Yaskawa INFORM job: SKRZYNIA_5040_180_STOPNI_10BR.JBI

/JOB
//NAME SKRZYNIA_5040_180_STOPNI_10BR
///FOLDERNAME 02-SKRZYNIE_JOBS
//POS
///NPOS 329,329,0,22,0,0
///TOOL 0
///POSTYPE PULSE
///PULSE
C00000=-21231,-51303,42314,2367,6591,-1439
C00001=-12854,-61498,-6635,149088,-29435,16513
C00002=84284,-61498,-6635,149088,14842,16513
C00003=84426,-61498,-62039,149088,14842,16513
C00004=84426,-61498,-83719,149088,14842,16513
C00005=79414,-27317,-83719,149088,18958,2543
C00006=69654,-19285,-77591,161600,-10201,-10832
C00007=70169,-17945,-76482,160305,-10504,-10321
C00008=68101,-15975,-74811,167053,-10620,-13110
C00009=69917,-14828,-73813,161695,-10968,-10930
C00010=70169,-17945,-76482,160305,-10504,-10321
C00011=40079,-25830,-61904,72398,37828,17494
C00012=40079,-25830,-61904,72398,37828,17494
C00013=38824,-23395,-60038,72349,38727,17731
C00014=41545,-22667,-59464,70826,37145,18191
C00015=40079,-25830,-61904,72398,37828,17494
C00016=62247,-7095,-69897,102362,7855,12255
C00017=53704,-22919,-41820,136356,29967,-7241
C00018=40577,-31455,-39147,101508,36831,1521
C00019=40669,-23760,-31845,100563,36582,2074
C00020=41101,-23552,-31684,100574,36285,2055
C00021=39898,-21530,-30092,99854,36985,2518
C00022=41920,-21198,-29826,100065,35629,2328
C00023=41101,-23552,-31684,100574,36285,2055
C00024=40577,-31455,-39147,101508,36831,1521
C00025=45746,-39048,-62846,85420,33792,9363
C00026=93007,-60609,-51405,156585,32340,-40977
C00027=83918,-61953,-48743,149551,29621,-25735
C00028=40577,-31455,-39147,101508,36831,1521
C00029=63645,-11488,-68603,127053,9270,213
C00030=57886,960,-43515,148211,29579,-11223
C00031=58100,6617,-53508,135301,20179,-4597
C00032=58076,11581,-47409,136064,20541,-4974
C00033=56683,13582,-44848,135736,21192,-4491
C00034=57911,14088,-44192,136506,20851,-5156
C00035=58076,11581,-47409,136064,20541,-4974
C00036=58100,6617,-53508,135301,20179,-4597
C00037=57886,960,-43515,148211,29579,-11223
C00038=63645,-11488,-68603,127053,9270,213
C00039=46424,-32589,-51504,107545,30005,2440
C00040=46670,-25209,-46239,104499,29210,4073
C00041=45428,-23318,-44777,103595,29873,4669
C00042=46971,-23118,-44620,103792,28881,4430
C00043=46670,-25209,-46239,104499,29210,4073
C00044=44789,-32224,-51260,106964,30993,2875
C00045=42092,-32720,-44065,59648,38266,12707
C00046=43496,-26383,-41044,56137,38810,14761
C00047=42389,-24633,-39725,56307,39660,14725
C00048=44413,-24250,-39432,55137,38557,15308
C00049=43496,-26383,-41044,56137,38810,14761
C00050=44564,-32742,-56962,40463,46428,19920
C00051=40345,-33419,-45947,59645,39680,12787
C00052=90538,-65158,-52413,145953,6697,-22013
C00053=90538,-65158,-52413,145953,6697,-22013
C00054=86028,-64310,-60026,34123,6588,25352
C00055=40577,-31455,-39147,101508,36831,1521
C00056=59968,-20268,-35682,154489,33643,-14406
C00057=58485,-14292,-30532,152791,33122,-13346
C00058=56876,-12305,-28713,151388,33319,-12442
C00059=58661,-11495,-27956,152741,32764,-13330
C00060=58485,-14292,-30532,152791,33122,-13346
C00061=59968,-20268,-35682,154489,33643,-14406
C00062=40577,-31455,-39147,101508,36831,1521
C00063=40577,-27956,-24714,110033,39226,-3600
C00064=40832,-22290,-20525,108598,38533,-2722
C00065=39477,-20111,-18797,107655,39231,-2172
C00066=41591,-19772,-18521,108272,37862,-2511
C00067=40832,-22290,-20525,108598,38533,-2722
C00068=40577,-31455,-39147,101508,36831,1521
C00069=86028,-64310,-60026,34123,6588,25352
C00070=86028,-64310,-60026,57978,24772,25352
C00071=86028,-64309,-60028,57978,24769,25352
C00072=40577,-31455,-39147,101508,36831,1521
C00073=40577,-31455,-39147,101508,36831,1521
C00074=41094,-24086,-28510,103808,36979,148
C00075=39566,-21578,-26552,102813,37826,761
C00076=41385,-20827,-24026,104651,36978,-353
C00077=41094,-24086,-28510,103808,36979,148
C00078=37787,-19718,1186,119438,46446,-9893
C00079=45975,-24882,-879,104701,32906,-9183
C00080=73009,-53529,-38439,45960,15190,15723
C00081=45844,-59376,-6382,28358,16063,-8083
C00082=0,-52280,40443,0,6876,0
C00083=-681,-52632,38645,-5695,5489,-631
C00084=-17840,-61498,-6635,-149088,-29435,-16513
C00085=-84284,-61498,-6635,-149088,14842,-16513
C00086=-84426,-61498,-62039,-149088,14842,-16513
C00087=-84426,-61498,-83719,-149088,14842,-16513
C00088=-79414,-27317,-83719,-149088,18958,-2543
C00089=-69654,-19285,-77591,-161600,-10201,10832
C00090=-70169,-17945,-76482,-160305,-10504,10321
C00091=-68828,-16679,-75416,-164694,-10564,12135
C00092=-70730,-15407,-74323,-159180,-10987,9897
C00093=-70169,-17945,-76482,-160305,-10504,10321
C00094=-69654,-19285,-77591,-161600,-10201,10832
C00095=-79414,-27317,-83719,-149088,18958,-2543
C00096=-79414,-27317,-83719,-149088,18958,-2543
C00097=-83351,-27062,-60322,-167360,37385,6517
C00098=-83351,-27062,-60322,-167360,37385,23281
C00099=-45097,-23850,-79932,-76262,26943,-22849
C00100=-48253,-15729,-73342,-71138,25693,-24842
C00101=-50302,-13076,-73239,-65836,25323,-27140
C00102=-49401,-11675,-71961,-66260,25816,-27133
C00103=-50608,-11574,-71867,-65226,25249,-27391
C00104=-49660,-13361,-73494,-66442,25615,-26975
C00105=-48242,-21102,-77802,-73044,25430,-23851
C00106=-42432,-29691,-46140,-101591,34194,-3953
C00107=-39561,-32409,-42051,-71473,38885,-9254
C00108=-41445,-24166,-34417,-69795,37942,-10196
C00109=-41357,-25431,-35380,-70168,37910,-9978
C00110=-40141,-23420,-33843,-70026,38836,-10113
C00111=-41944,-23213,-33680,-69384,37685,-10425
C00112=-41357,-25431,-35380,-70168,37910,-9978
C00113=-39561,-32409,-42051,-71473,38885,-9254
C00114=-81019,-65479,-53594,-111483,16801,11860
C00115=-83918,-61953,-48743,-149551,29621,25735
C00116=-40577,-31455,-39147,-101508,36831,-1521
C00117=-49519,-25509,-75942,-81549,24001,-19130
C00118=-42138,-12822,-51897,-114220,37124,-2825
C00119=-42418,-8239,-63642,-99180,32968,-11424
C00120=-44218,-2315,-57613,-98259,31965,-11515
C00121=-43448,-826,-56017,-98426,32361,-11601
C00122=-45030,-456,-55613,-98008,31536,-11462
C00123=-44218,-2315,-57613,-98259,31965,-11515
C00124=-42418,-8239,-63642,-99180,32968,-11424
C00125=-46424,-32589,-51504,-107545,30005,-2440
C00126=-47664,-24599,-45775,-104463,28531,-3999
C00127=-46974,-23582,-44988,-103952,28901,-4330
C00128=-48737,-23213,-44698,-104162,27760,-4069
C00129=-47664,-24599,-45775,-104463,28531,-3999
C00130=-44789,-32224,-51260,-106964,30993,-2875
C00131=-52916,-26599,-39279,-28650,42861,-21372
C00132=-54590,-19092,-33239,-26753,43640,-22510
C00133=-53867,-18183,-32472,-27186,44006,-22274
C00134=-55270,-17868,-32204,-26176,43615,-22844
C00135=-54590,-19092,-33239,-26753,43640,-22510
C00136=-51388,-27442,-41316,-29309,44045,-21030
C00137=-62081,-38823,-47091,-30795,32483,-22364
C00138=-86028,-64310,-60024,-34123,6590,-25350
C00139=-86028,-64310,-60026,-34123,6588,-25352
C00140=-86028,-64310,-60026,-34123,6588,-25352
C00141=-40577,-31455,-39147,-101508,36831,-1521
C00142=-46190,-29637,-41119,-118468,33777,2449
C00143=-49093,-22876,-34875,-118816,31686,2771
C00144=-47416,-20516,-32984,-117411,32403,1908
C00145=-48747,-20402,-32891,-117991,31622,2296
C00146=-49093,-22876,-34875,-118816,31686,2771
C00147=-46494,-29071,-39687,-120554,34221,3238
C00148=-39561,-32409,-42051,-71473,38885,-9254
C00149=-39561,-29125,-27808,-80306,37382,-3940
C00150=-43436,-23752,-23915,-78119,34960,-5282
C00151=-41521,-20874,-21664,-77573,36353,-5586
C00152=-43032,-20790,-21597,-77323,35339,-5740
C00153=-43436,-23752,-23915,-78119,34960,-5282
C00154=-39561,-32409,-42051,-71473,38885,-9254
C00155=-86028,-64310,-60026,-34123,6588,-25352
C00156=-86028,-64310,-60026,-57978,24772,-25352
C00157=-86028,-64309,-60028,-57978,24769,-25352
C00158=-40577,-28664,-27343,-108630,38732,2744
C00159=-40577,-31455,-39147,-101508,36831,-1521
C00160=-43516,-21710,-22385,-107479,36200,2021
C00161=-42168,-19388,-19611,-107236,37117,1884
C00162=-43632,-19706,-21236,-106626,35874,1517
C00163=-43516,-21710,-22385,-107479,36200,2021
C00164=-37787,-19718,1186,-119438,46446,9893
C00165=-42073,-20304,2487,-100625,34839,7554
C00166=-73009,-40277,-6382,-95546,11240,8083
C00167=-45844,-59376,-6382,-28358,16063,8083
C00168=0,-52280,40443,0,6876,0
C00169=0,-52280,40443,0,6876,0
C00170=0,-52280,40443,0,6876,0
C00171=17840,-61498,-6635,149088,-29435,16513
C00172=84284,-61498,-6635,149088,14842,16513
C00173=84426,-61498,-62039,149088,14842,16513
C00174=84426,-61498,-83719,149088,14842,16513
C00175=79414,-27317,-83719,149088,18958,2543
C00176=69654,-19285,-77591,161600,-10201,-10832
C00177=76421,-10554,-96109,158804,-42582,-3780
C00178=72151,-15398,-68153,108866,-8938,34672
C00179=72146,-15003,-68876,113258,-9266,32587
C00180=76421,-10554,-96109,158804,-42582,-3780
C00181=34693,-20653,-55351,82826,43754,17424
C00182=36026,-17403,-55626,79704,43213,19225
C00183=36110,-16271,-60816,75273,43939,22119
C00184=33117,-22954,-57201,83762,44711,17076
C00185=44072,-25282,-29267,59074,37137,11149
C00186=35613,-12237,-16796,64347,49532,7989
C00187=35669,-10629,-9632,67221,48090,5904
C00188=43298,-18069,-12230,66933,34938,6545
C00189=45101,-28611,-34216,51905,38288,13313
C00190=86972,-59792,-47806,52261,11911,13502
C00191=84284,-61498,-6635,149088,14842,16513
C00192=17840,-61498,-6635,149088,-29435,16513
C00193=0,-52280,40443,0,6876,0
C00194=-84284,-61498,-6635,-149088,14842,-16513
C00195=-84426,-61498,-62039,-149088,14842,-16513
C00196=-34728,-20635,-55362,-82794,43735,-17439
C00197=-36397,-18395,-56469,-79733,42961,-19136
C00198=-36362,-17151,-61599,-75273,43766,-22060
C00199=-33152,-22936,-57213,-83730,44691,-17092
C00200=-40586,-30782,-66310,-80775,34854,-15242
C00201=-40692,-30585,-47134,-93878,35604,-6100
C00202=-40870,-31947,-42232,-63836,39356,-11267
C00203=-40932,-24208,-34937,-62959,39653,-11802
C00204=-45435,-25401,-38781,-45915,41942,-16635
C00205=-39287,-15996,-33256,-50997,52191,-14482
C00206=-39287,-15215,-27013,-53302,49993,-12721
C00207=-47238,-24614,-37591,-45025,40897,-17096
C00208=-47977,-29416,-47116,-37884,44778,-19458
C00209=-89911,-63274,-62690,-19483,20389,-28477
C00210=-84284,-61498,-6635,-149088,14842,-16513
C00211=-17840,-61498,-6635,-149088,-29435,-16513
C00212=-2124,-53377,34839,-17747,2554,-1966
C00213=0,-52279,40442,0,6873,-1
C00214=65212,-60046,-8049,104848,-4690,-17864
C00215=40577,-31455,-39147,101508,36831,1521
C00216=38935,-8667,-59866,96806,37491,11641
C00217=39872,-3948,-62200,89905,36425,15493
C00218=40123,-1398,-59509,89712,36292,15545
C00219=40076,1432,-63122,83669,36365,19101
C00220=39872,-3948,-62200,89905,36425,15493
C00221=38788,-10415,-65666,93500,37192,13644
C00222=38494,-13737,-58620,102504,38775,8306
C00223=46486,-25212,-81916,68038,29584,25152
C00224=40809,-36068,-61713,64442,39202,15742
C00225=42276,-26166,-36634,93086,33999,4511
C00226=42397,-24236,-35180,92449,33874,4870
C00227=42456,-24928,-41878,86540,33672,8224
C00228=42276,-26166,-36634,93086,33999,4511
C00229=39142,-35579,-61405,65081,40271,15536
C00230=56371,-25371,-52824,18615,54374,25524
C00231=56370,-25165,-46553,19645,50450,24711
C00232=56832,-16031,-39063,18899,51967,25222
C00233=56804,-15583,-32487,20072,48035,24353
C00234=56370,-25165,-46553,19645,50450,24711
C00235=57699,-31993,-47488,30685,42383,20627
C00236=72028,-54906,-32140,129304,10545,-19932
C00237=68553,-57528,-19846,116818,2770,-18873
C00238=80051,-74607,19733,-8233,-9721,30787
C00239=0,-52279,40442,0,6873,1
C00240=-65212,-60046,-8049,-104848,-4690,17864
C00241=-65212,-60046,-8049,-104848,-4690,17864
C00242=-38865,-30967,-34224,-83703,38027,-4479
C00243=-46136,-6939,-46632,-121706,34309,84
C00244=-46867,-3267,-49648,-115679,31344,-3160
C00245=-48114,-333,-46510,-115722,30691,-2892
C00246=-48219,1611,-50657,-109137,28744,-6443
C00247=-46867,-3267,-49648,-115679,31344,-3160
C00248=-46241,-9247,-52869,-118634,32829,-1638
C00249=-45976,-11042,-44788,-126297,37070,2732
C00250=-52833,-24736,-69580,-100186,20368,-10781
C00251=-41290,-34357,-47396,-89099,34671,-6127
C00252=-41655,-21075,-14083,-101384,36064,2719
C00253=-43548,-19389,-12736,-101518,34735,2718
C00254=-43554,-21360,-20853,-95828,33898,-537
C00255=-41655,-21075,-14083,-101384,36064,2719
C00256=-39902,-32831,-41704,-71274,37363,-9142
C00257=-59997,-20337,-29256,-15458,45038,-24823
C00258=-49653,-28135,-37805,-37523,39695,-18391
C00259=-43199,-13906,-27547,-44351,51052,-15347
C00260=-43351,-12703,-20152,-46774,48118,-13551
C00261=-49653,-28135,-37805,-37523,39695,-18391
C00262=-55865,-33769,-26948,-46240,25044,-14477
C00263=-87889,-52133,-21276,-78165,-5410,-1028
C00264=0,-52279,40442,0,6873,1
C00265=1,-52278,40440,0,6869,2
C00266=71244,-62242,-42760,28259,6636,20995
C00267=86028,-64310,-60026,34123,6588,25352
C00268=40577,-31455,-39147,101508,36831,1521
C00269=59968,-20268,-35682,154489,33643,-14406
C00270=58485,-13865,-27025,153905,35067,-13980
C00271=58455,-11202,-24562,153724,34784,-13877
C00272=58575,-12016,-31397,151462,30972,-12614
C00273=58485,-13865,-27025,153905,35067,-13980
C00274=59968,-20268,-35682,154489,33643,-14406
C00275=40577,-31455,-39147,101508,36831,1521
C00276=39533,-29159,-27906,80257,37406,3969
C00277=37605,-21741,-8857,99005,39903,-3768
C00278=39778,-16633,-4738,98441,38266,-3268
C00279=39778,-19203,-13530,93410,37627,-246
C00280=39876,-23449,-23758,78420,37382,5067
C00281=40577,-31455,-39147,101508,36831,1521
C00282=86028,-64310,-60026,34123,6588,25352
C00283=71244,-62242,-42760,28259,6636,20995
C00284=1,-52278,40440,0,6869,2
C00285=1,-52278,40440,0,6869,2
C00286=-71244,-62242,-42760,-28259,6636,-20995
C00287=-86028,-64310,-60026,-34123,6588,-25352
C00288=-40577,-31455,-39147,-101508,36831,-1521
C00289=-59968,-20268,-35682,-154489,33643,14406
C00290=-58485,-13865,-27025,-153905,35067,13980
C00291=-60457,-10469,-23870,-155260,34234,14880
C00292=-60514,-11164,-30597,-153048,30384,13645
C00293=-58485,-13865,-27025,-153905,35067,13980
C00294=-59968,-20268,-35682,-154489,33643,14406
C00295=-40577,-31455,-39147,-101508,36831,-1521
C00296=-39561,-29149,-27902,-80249,37387,-3974
C00297=-37632,-21733,-8858,-99006,39884,3767
C00298=-42115,-16101,-4294,-98986,36705,3442
C00299=-42200,-18704,-13124,-93672,35977,314
C00300=-39902,-23438,-23752,-78411,37365,-5072
C00301=-39561,-32409,-42051,-71473,38885,-9254
C00302=-86028,-64310,-60026,-34123,6588,-25352
C00303=-71244,-62242,-42760,-28259,6636,-20995
C00304=-1,-52278,40440,0,6869,-2
C00305=2,-52272,40438,1,6859,6
C00306=86028,-64309,-60028,57978,24769,25352
C00307=40577,-31455,-39147,101508,36831,1521
C00308=41094,-22734,-22712,107351,37942,-1964
C00309=41295,-19722,-19354,107466,37828,-2032
C00310=41253,-21899,-28956,101408,36344,1561
C00311=41094,-22306,-21006,108327,38251,-2553
C00312=37787,-19718,1186,119438,46446,-9893
C00313=73009,-40734,-7449,93649,11189,-7175
C00314=45844,-59376,-6382,28358,16063,-8083
C00315=0,-52280,40443,0,6876,0
C00316=-2,-52272,40438,-1,6859,-6
C00317=-86028,-64309,-60028,-57978,24769,-25352
C00318=-40577,-30748,-35855,-103638,37302,-257
C00319=-40400,-24560,-25747,-102945,37769,566
C00320=-40181,-24927,-30789,-96759,37058,-2330
C00321=-42523,-20980,-24961,-98936,35699,-1187
C00322=-42523,-22298,-31586,-94154,35106,-3962
C00323=-42312,-27031,-36420,-94462,35277,-3790
C00324=-37787,-19718,1186,-119438,46446,9893
C00325=-73009,-37989,-1068,-104580,11683,12408
C00326=-45844,-59376,-6382,-28358,16063,8083
C00327=0,-52280,40443,0,6876,0
C00328=0,-52279,40442,1,6873,0
BC00000=467225
BC00001=513669
BC00002=494109
BC00003=467540
BC00004=467540
BC00005=467540
BC00006=467540
BC00007=467540
BC00008=467540
BC00009=467540
BC00010=467540
BC00011=478876
BC00012=478876
BC00013=478876
BC00014=478876
BC00015=478876
BC00016=566479
BC00017=516375
BC00018=516375
BC00019=516375
BC00020=516375
BC00021=516375
BC00022=516375
BC00023=516375
BC00024=516375
BC00025=488496
BC00026=488496
BC00027=675626
BC00028=675626
BC00029=717870
BC00030=717870
BC00031=717870
BC00032=717870
BC00033=717870
BC00034=717870
BC00035=717870
BC00036=717870
BC00037=717870
BC00038=717870
BC00039=686402
BC00040=686402
BC00041=686402
BC00042=686402
BC00043=686402
BC00044=686402
BC00045=673769
BC00046=686402
BC00047=686402
BC00048=686402
BC00049=686402
BC00050=686402
BC00051=641577
BC00052=641414
BC00053=760541
BC00054=849627
BC00055=849627
BC00056=849627
BC00057=849627
BC00058=849627
BC00059=849627
BC00060=849627
BC00061=849627
BC00062=849627
BC00063=849627
BC00064=849627
BC00065=849627
BC00066=849627
BC00067=849627
BC00068=849627
BC00069=849627
BC00070=849627
BC00071=998332
BC00072=998017
BC00073=1002378
BC00074=995834
BC00075=995834
BC00076=993496
BC00077=995834
BC00078=965704
BC00079=965704
BC00080=965704
BC00081=879640
BC00082=828403
BC00083=518986
BC00084=509920
BC00085=467540
BC00086=467540
BC00087=467540
BC00088=467540
BC00089=467540
BC00090=467540
BC00091=467540
BC00092=467540
BC00093=467540
BC00094=467540
BC00095=467540
BC00096=550011
BC00097=521167
BC00098=520352
BC00099=535759
BC00100=535759
BC00101=535757
BC00102=535757
BC00103=535757
BC00104=535757
BC00105=535757
BC00106=485653
BC00107=485653
BC00108=485653
BC00109=485653
BC00110=485653
BC00111=485653
BC00112=485653
BC00113=485653
BC00114=485653
BC00115=675626
BC00116=675626
BC00117=687148
BC00118=687148
BC00119=687148
BC00120=687148
BC00121=687148
BC00122=687148
BC00123=687148
BC00124=687148
BC00125=686402
BC00126=686401
BC00127=686401
BC00128=686401
BC00129=686401
BC00130=686402
BC00131=655680
BC00132=655680
BC00133=655680
BC00134=655680
BC00135=655680
BC00136=655680
BC00137=643721
BC00138=659181
BC00139=817027
BC00140=849627
BC00141=849627
BC00142=818905
BC00143=818905
BC00144=818905
BC00145=818905
BC00146=818905
BC00147=818905
BC00148=818905
BC00149=818905
BC00150=818905
BC00151=818905
BC00152=818905
BC00153=818905
BC00154=818905
BC00155=849627
BC00156=849627
BC00157=983499
BC00158=985574
BC00159=996021
BC00160=990664
BC00161=989585
BC00162=991221
BC00163=990664
BC00164=965704
BC00165=965704
BC00166=946312
BC00167=879640
BC00168=828403
BC00169=639407
BC00170=514217
BC00171=512528
BC00172=467540
BC00173=467540
BC00174=467540
BC00175=467540
BC00176=467540
BC00177=467540
BC00178=467538
BC00179=467538
BC00180=467540
BC00181=489674
BC00182=489674
BC00183=489674
BC00184=489674
BC00185=454931
BC00186=454931
BC00187=454931
BC00188=454931
BC00189=454931
BC00190=454931
BC00191=467540
BC00192=515629
BC00193=504733
BC00194=467540
BC00195=467540
BC00196=489675
BC00197=489675
BC00198=489675
BC00199=489675
BC00200=489675
BC00201=477973
BC00202=477973
BC00203=477973
BC00204=462612
BC00205=462612
BC00206=462612
BC00207=462612
BC00208=462612
BC00209=462612
BC00210=467540
BC00211=497858
BC00212=502748
BC00213=574255
BC00214=557840
BC00215=654869
BC00216=687148
BC00217=687148
BC00218=687148
BC00219=687148
BC00220=687148
BC00221=687148
BC00222=687148
BC00223=687148
BC00224=655680
BC00225=655680
BC00226=655680
BC00227=655680
BC00228=655680
BC00229=655680
BC00230=655680
BC00231=655680
BC00232=655680
BC00233=655680
BC00234=655680
BC00235=638520
BC00236=608041
BC00237=573428
BC00238=574255
BC00239=574255
BC00240=626137
BC00241=536464
BC00242=650227
BC00243=687148
BC00244=687148
BC00245=687148
BC00246=687148
BC00247=687148
BC00248=687148
BC00249=687148
BC00250=687148
BC00251=655680
BC00252=624958
BC00253=624958
BC00254=624958
BC00255=624958
BC00256=624958
BC00257=624958
BC00258=655680
BC00259=655680
BC00260=655680
BC00261=655680
BC00262=605110
BC00263=576379
BC00264=574255
BC00265=574254
BC00266=802302
BC00267=849627
BC00268=849627
BC00269=849627
BC00270=849627
BC00271=849627
BC00272=849627
BC00273=849627
BC00274=849627
BC00275=849627
BC00276=818905
BC00277=818905
BC00278=818905
BC00279=818905
BC00280=818905
BC00281=849627
BC00282=849627
BC00283=802302
BC00284=652677
BC00285=652677
BC00286=802302
BC00287=849627
BC00288=849627
BC00289=849627
BC00290=849627
BC00291=849629
BC00292=849627
BC00293=849627
BC00294=849627
BC00295=849627
BC00296=818905
BC00297=818905
BC00298=818905
BC00299=818905
BC00300=818905
BC00301=818905
BC00302=849627
BC00303=802302
BC00304=652677
BC00305=780547
BC00306=993116
BC00307=996061
BC00308=994027
BC00309=992881
BC00310=994683
BC00311=992390
BC00312=965704
BC00313=946311
BC00314=879640
BC00315=828403
BC00316=780547
BC00317=988063
BC00318=993111
BC00319=990227
BC00320=995173
BC00321=992391
BC00322=992391
BC00323=992391
BC00324=965704
BC00325=939357
BC00326=879640
BC00327=828403
BC00328=644864
///POSTYPE BASE
///RECTAN
///RCONF 1,0,0,0,0,0,0,0,0,0,0,0,0,0,0,0,0,0,0,0,0,0,0,0
P00006=0.046,-2.112,7.779,0.0000,0.0000,0.0000
///RCONF 0,0,0,0,0,0,0,0,0,0,0,0,0,0,0,0,0,0,0,0,0,0,0,0
P00056=0.000,0.000,5.000,0.0000,0.0000,0.0000
///RCONF 1,0,0,0,0,0,0,0,0,0,0,0,0,0,0,0,0,0,0,0,0,0,0,0
P00300=-0.036,-1.505,2.318,0.0000,0.0000,0.0000
P00301=0.046,-2.112,7.779,0.0000,0.0000,0.0000
///RCONF 0,0,0,0,0,0,0,0,0,0,0,0,0,0,0,0,0,0,0,0,0,0,0,0
P00302=0.052,-2.937,-4.426,0.0000,0.0000,0.0000
P00303=-0.004,-1.437,-4.584,0.0000,0.0000,0.0000
P00304=0.028,-1.666,-4.234,0.0000,0.0000,0.0000
P00305=-0.003,-1.920,-3.501,0.0000,0.0000,0.0000
P00306=0.015,-2.252,-3.054,0.0000,0.0000,0.0000
P00307=0.019,-2.151,-5.077,0.0000,0.0000,0.0000
P00308=-0.003,-2.092,-4.888,0.0000,0.0000,0.0000
P00309=-0.040,-2.205,-4.992,0.0000,0.0000,0.0000
P00350=11.519,-0.008,1.149,0.0000,0.0000,0.0000
P00351=13.563,-0.027,-0.653,0.0000,0.0000,0.0000
P00352=13.252,-0.027,-0.827,0.0000,0.0000,0.0000
P00353=10.971,-0.082,0.776,0.0000,0.0000,0.0000
P00354=-0.024,2.508,-1.824,0.0000,0.0000,0.0000
P00355=-0.001,2.528,-1.131,0.0000,0.0000,0.0000
P00356=-0.034,2.921,-0.262,0.0000,0.0000,0.0000
P00357=0.003,3.386,-0.091,0.0000,0.0000,0.0000
P00358=0.014,3.037,-0.020,0.0000,0.0000,0.0000
P00359=-0.005,2.731,0.912,0.0000,0.0000,0.0000
//INST
///DATE 2024/05/14 10:01
///ATTR SC,RW
///GROUP1 RB1,BS1
NOP
CALL JOB:MOVE_INTO_TUNNEL
MOVJ C00000 BC00000 VJ=10.00
MOVJ C00001 BC00001 VJ=10.00
MOVJ C00002 BC00002 VJ=10.00
MOVJ C00003 BC00003 VJ=10.00
MOVJ C00004 BC00004 VJ=10.00
MOVJ C00005 BC00005 VJ=10.00
MOVJ C00006 BC00006 VJ=10.00
'------------------------
'W29.2
'------------------------
MOVL C00007 BC00007 V=66.7 PL=0
REFP 3 C00008 BC00008
CALL JOB:SEARCH-R1
IMOV P0056 V=23.0
SET P0300 P0006
SFTON P0300
REFP 3 C00009 BC00009
CALL JOB:SEARCH-R1
SET P0300 P0006
SFTON P0300
MOVL C00010 BC00010 V=66.7 PL=0
SFTOF
'PRZEJAZD
MOVL C00011 BC00011 V=500.0
'------------------------
'W63.5
'------------------------
MOVL C00012 BC00012 V=66.7 PL=0
REFP 3 C00013 BC00013
CALL JOB:SEARCH-R1
IMOV P0056 V=23.0 PL=0
SET P0301 P0006
SFTON P0301
REFP 3 C00014 BC00014
CALL JOB:SEARCH-R1
SET P0301 P0006
SFTON P0301
MOVL C00015 BC00015 V=66.7 PL=0
SFTOF
GETE D040 P0301 (1)
GETE D041 P0301 (2)
GETE D042 P0301 (3)
SETE P0302 (1) D040
SETE P0302 (2) D041
SETE P0302 (3) D042
COMM 'PRZEJAZD
COMM MOVL C00016 BC00016 V=500.0
COMM MOVL C00017 BC00017 V=500.0
COMM MOVL C00018 BC00018 V=500.0
COMM MOVL C00019 BC00019 V=500.0
COMM '------------------------
COMM 'W29.8
COMM '------------------------
COMM MOVL C00020 BC00020 V=66.7 PL=0
COMM REFP 3 C00021 BC00021
COMM CALL JOB:SEARCH-R1
COMM IMOV P0056 V=23.0 PL=0
COMM SET P0302 P0006
COMM SFTON P0302
COMM REFP 3 C00022 BC00022
COMM CALL JOB:SEARCH-R1
COMM SET P0302 P0006
COMM SFTON P0302
COMM MOVL C00023 BC00023 V=66.7 PL=0
COMM SFTOF
COMM MOVL C00024 BC00024 V=500.0
COMM 'PRZEJAZD
MOVL C00025 BC00025 V=500.0
MOVJ C00026 BC00026 VJ=10.00
MOVJ C00027 BC00027 VJ=10.00
MOVL C00028 BC00028 V=500.0
MOVL C00029 BC00029 V=500.0
MOVL C00030 BC00030 V=500.0
MOVL C00031 BC00031 V=500.0
'------------------------
'W29.11
'------------------------
MOVL C00032 BC00032 V=66.7 PL=0
REFP 3 C00033 BC00033
CALL JOB:SEARCH-R1
IMOV P0056 V=23.0 PL=0
SET P0303 P0006
SFTON P0303
REFP 3 C00034 BC00034
CALL JOB:SEARCH-R1
SET P0303 P0006
SFTON P0303
MOVL C00035 BC00035 V=66.7 PL=0
SFTOF
'PRZEJAZD
MOVL C00036 BC00036 V=500.0
MOVL C00037 BC00037 V=500.0
MOVL C00038 BC00038 V=500.0
MOVL C00039 BC00039 V=500.0
'------------------------
'W29.14
'------------------------
MOVL C00040 BC00040 V=66.7 PL=0
REFP 3 C00041 BC00041
CALL JOB:SEARCH-R1
IMOV P0056 V=23.0 PL=0
SET P0304 P0006
SFTON P0304
REFP 3 C00042 BC00042
CALL JOB:SEARCH-R1
SET P0304 P0006
SFTON P0304
MOVL C00043 BC00043 V=66.7 PL=0
SFTOF
'PRZEJAZD
MOVL C00044 BC00044 V=500.0
MOVL C00045 BC00045 V=500.0
'------------------------
'W63.17
'------------------------
MOVL C00046 BC00046 V=166.7 PL=0
REFP 3 C00047 BC00047
CALL JOB:SEARCH-R1
IMOV P0056 V=23.0 PL=0
SET P0305 P0006
SFTON P0305
REFP 3 C00048 BC00048
CALL JOB:SEARCH-R1
SET P0305 P0006
SFTON P0305
MOVL C00049 BC00049 V=66.7 PL=0
SFTOF
'PRZEJAZD
MOVL C00050 BC00050 V=500.0
MOVJ C00051 BC00051 VJ=10.00
MOVJ C00052 BC00052 VJ=10.00
MOVJ C00053 BC00053 VJ=30.00
MOVJ C00054 BC00054 VJ=30.00
MOVL C00055 BC00055 V=500.0
MOVL C00056 BC00056 V=500.0
'------------------------
'W63.20
'------------------------
MOVL C00057 BC00057 V=66.7 PL=0
REFP 3 C00058 BC00058
CALL JOB:SEARCH-R1
IMOV P0056 V=23.0 PL=0
SET P0306 P0006
SFTON P0306
REFP 3 C00059 BC00059
CALL JOB:SEARCH-R1
SET P0306 P0006
SFTON P0306
MOVL C00060 BC00060 V=66.7 PL=0
SFTOF
'PRZEJAZD
MOVL C00061 BC00061 V=500.0
MOVL C00062 BC00062 V=500.0
MOVL C00063 BC00063 V=500.0
'------------------------
'W63.23
'------------------------
MOVL C00064 BC00064 V=66.7 PL=0
REFP 3 C00065 BC00065
CALL JOB:SEARCH-R1
IMOV P0056 V=23.0 PL=0
SET P0307 P0006
SFTON P0307
REFP 3 C00066 BC00066
CALL JOB:SEARCH-R1
SET P0307 P0006
SFTON P0307
MOVL C00067 BC00067 V=66.7 PL=0
SFTOF
'PRZEJAZD
'BRAK 29.26
'BRAK 29.26
'BRAK 29.26
GETE D040 P0307 (1)
GETE D041 P0307 (2)
GETE D042 P0307 (3)
SETE P0308 (1) D040
SETE P0308 (2) D041
SETE P0308 (3) D042
'BRAK 29.26
'BRAK 29.26
'BRAK 29.26
MOVL C00068 BC00068 V=500.0
MOVL C00069 BC00069 V=500.0
MOVL C00070 BC00070 V=500.0
MOVL C00071 BC00071 V=500.0
MOVL C00072 BC00072 V=500.0
MOVL C00073 BC00073 V=500.0
'------------------------
'W29.29
'------------------------
MOVL C00074 BC00074 V=66.7 PL=0
REFP 3 C00075 BC00075
CALL JOB:SEARCH-R1
IMOV P0056 V=23.0 PL=0
SET P0309 P0006
SFTON P0309
REFP 3 C00076 BC00076
CALL JOB:SEARCH-R1
SET P0309 P0006
SFTON P0309
MOVL C00077 BC00077 V=66.7 PL=0
SFTOF
'PRZEJAZD
MOVL C00078 BC00078 V=500.0
'PRZEJAZD
MOVL C00079 BC00079 V=500.0
MOVJ C00080 BC00080 VJ=10.00
MOVJ C00081 BC00081 VJ=10.00
MOVJ C00082 BC00082 VJ=20.00
MOVJ C00083 BC00083 VJ=30.00
MOVJ C00084 BC00084 VJ=20.00
MOVJ C00085 BC00085 VJ=10.00
MOVJ C00086 BC00086 VJ=20.00
MOVJ C00087 BC00087 VJ=20.00
MOVJ C00088 BC00088 VJ=20.00
MOVJ C00089 BC00089 VJ=20.00
'------------------------
'W28.2
'------------------------
MOVL C00090 BC00090 V=66.7 PL=0
REFP 3 C00091 BC00091
CALL JOB:SEARCH-R1
IMOV P0056 V=23.0
SET P0350 P0006
SFTON P0350
REFP 3 C00092 BC00092
CALL JOB:SEARCH-R1
SET P0350 P0006
SFTON P0350
MOVL C00093 BC00093 V=66.7 PL=0
SFTOF
'PRZEJAZD
MOVJ C00094 BC00094 VJ=10.00
MOVJ C00095 BC00095 VJ=10.00
MOVJ C00096 BC00096 VJ=10.00
MOVJ C00097 BC00097 VJ=10.00
MOVJ C00098 BC00098 VJ=10.00
MOVL C00099 BC00099 V=500.0
MOVL C00100 BC00100 V=500.0
'------------------------
'W62.5
'------------------------
MOVL C00101 BC00101 V=66.7 PL=0
REFP 3 C00102 BC00102
CALL JOB:SEARCH-R1
IMOV P0056 V=23.0 PL=0
SET P0351 P0006
SFTON P0351
REFP 3 C00103 BC00103
CALL JOB:SEARCH-R1
SET P0351 P0006
SFTON P0351
MOVL C00104 BC00104 V=66.7 PL=0
SFTOF
'PRZEJAZD
MOVL C00105 BC00105 V=500.0
MOVL C00106 BC00106 V=500.0
MOVL C00107 BC00107 V=500.0
MOVL C00108 BC00108 V=500.0
'------------------------
'W29.8
'------------------------
MOVL C00109 BC00109 V=66.7 PL=0
REFP 3 C00110 BC00110
CALL JOB:SEARCH-R1
IMOV P0056 V=23.0 PL=0
SET P0352 P0006
SFTON P0352
REFP 3 C00111 BC00111
CALL JOB:SEARCH-R1
SET P0352 P0006
SFTON P0352
MOVL C00112 BC00112 V=66.7 PL=0
SFTOF
MOVL C00113 BC00113 V=500.0
'PRZEJAZD
MOVL C00114 BC00114 V=500.0
MOVJ C00115 BC00115 VJ=20.00
MOVL C00116 BC00116 V=500.0
MOVL C00117 BC00117 V=500.0
MOVL C00118 BC00118 V=500.0
MOVL C00119 BC00119 V=500.0
'------------------------
'W29.11
'------------------------
MOVL C00120 BC00120 V=66.7 PL=0
REFP 3 C00121 BC00121
CALL JOB:SEARCH-R1
IMOV P0056 V=23.0 PL=0
SET P0353 P0006
SFTON P0353
REFP 3 C00122 BC00122
CALL JOB:SEARCH-R1
SET P0353 P0006
SFTON P0353
MOVL C00123 BC00123 V=66.7 PL=0
SFTOF
'PRZEJAZD
MOVL C00124 BC00124 V=500.0
MOVL C00125 BC00125 V=500.0
'------------------------
'W29.14
'------------------------
MOVL C00126 BC00126 V=66.7 PL=0
REFP 3 C00127 BC00127
CALL JOB:SEARCH-R1
IMOV P0056 V=23.0 PL=0
SET P0354 P0006
SFTON P0354
REFP 3 C00128 BC00128
CALL JOB:SEARCH-R1
SET P0354 P0006
SFTON P0354
MOVL C00129 BC00129 V=66.7 PL=0
SFTOF
'PRZEJAZD
MOVL C00130 BC00130 V=500.0
MOVL C00131 BC00131 V=500.0
'------------------------
'W63.17
'------------------------
MOVL C00132 BC00132 V=66.7 PL=0
REFP 3 C00133 BC00133
CALL JOB:SEARCH-R1
IMOV P0056 V=23.0 PL=0
SET P0355 P0006
SFTON P0355
REFP 3 C00134 BC00134
CALL JOB:SEARCH-R1
SET P0355 P0006
SFTON P0355
MOVL C00135 BC00135 V=66.7 PL=0
SFTOF
'PRZEJAZD
MOVL C00136 BC00136 V=500.0
MOVJ C00137 BC00137 VJ=10.00
MOVJ C00138 BC00138 VJ=10.00
MOVJ C00139 BC00139 VJ=10.00
MOVJ C00140 BC00140 VJ=10.00
MOVL C00141 BC00141 V=500.0
MOVL C00142 BC00142 V=500.0
'------------------------
'W62.20
'------------------------
MOVL C00143 BC00143 V=66.7 PL=0
REFP 3 C00144 BC00144
CALL JOB:SEARCH-R1
IMOV P0056 V=23.0 PL=0
SET P0356 P0006
SFTON P0356
REFP 3 C00145 BC00145
CALL JOB:SEARCH-R1
SET P0356 P0006
SFTON P0356
MOVL C00146 BC00146 V=66.7 PL=0
SFTOF
'PRZEJAZD
MOVL C00147 BC00147 V=500.0
MOVL C00148 BC00148 V=500.0
MOVL C00149 BC00149 V=500.0
'------------------------
'W63.23
'------------------------
MOVL C00150 BC00150 V=66.7 PL=0
REFP 3 C00151 BC00151
CALL JOB:SEARCH-R1
IMOV P0056 V=23.0 PL=0
SET P0357 P0006
SFTON P0357
REFP 3 C00152 BC00152
CALL JOB:SEARCH-R1
SET P0357 P0006
SFTON P0357
MOVL C00153 BC00153 V=66.7 PL=0
SFTOF
'PRZEJAZD
'BRAK 29.26
'BRAK 29.26
'BRAK 29.26
'BRAK 29.26
GETE D040 P0357 (1)
GETE D041 P0357 (2)
GETE D042 P0357 (3)
SETE P0358 (1) D040
SETE P0358 (2) D041
SETE P0358 (3) D042
'BRAK 29.26
'BRAK 29.26
MOVL C00154 BC00154 V=500.0
MOVL C00155 BC00155 V=500.0
MOVL C00156 BC00156 V=500.0
MOVL C00157 BC00157 V=500.0
MOVL C00158 BC00158 V=500.0
MOVL C00159 BC00159 V=500.0
'------------------------
'W29.29
'------------------------
MOVL C00160 BC00160 V=66.7 PL=0
REFP 3 C00161 BC00161
CALL JOB:SEARCH-R1
IMOV P0056 V=23.0 PL=0
SET P0359 P0006
SFTON P0359
REFP 3 C00162 BC00162
CALL JOB:SEARCH-R1
SET P0359 P0006
SFTON P0359
MOVL C00163 BC00163 V=66.7 PL=0
SFTOF
'PRZEJAZD
MOVL C00164 BC00164 V=500.0
'------------------------
'W29.32
'------------------------
'PRZEJAZD
MOVL C00165 BC00165 V=500.0
MOVJ C00166 BC00166 VJ=10.00
MOVJ C00167 BC00167 VJ=20.00
MOVJ C00168 BC00168 VJ=20.00
MOVJ C00169 BC00169 VJ=20.00
MOVJ C00170 BC00170 VJ=20.00
MOVJ C00171 BC00171 VJ=10.00
MOVJ C00172 BC00172 VJ=10.00
MOVJ C00173 BC00173 VJ=10.00
MOVJ C00174 BC00174 VJ=10.00
MOVJ C00175 BC00175 VJ=10.00
MOVJ C00176 BC00176 VJ=10.00
'------------------------
'W29.2
'------------------------
MOVL C00177 BC00177 V=500.0
SFTON P0300
MOVL C00178 BC00178 V=66.7 PL=0
MACRO1 MJ#(0) ARGF24
MOVL C00179 BC00179 V=10.8
ARCOF
SFTOF
MOVL C00180 BC00180 V=500.0
'PRZEJAZD
'------------------------
'W63.5
'------------------------
MOVL C00181 BC00181 V=500.0
SFTON P0301
MOVL C00182 BC00182 V=66.7 PL=0
MACRO1 MJ#(0) ARGF24
ARCON
MOVL C00183 BC00183 V=10.0
ARCOF
SFTOF
MOVL C00184 BC00184 V=500.0
'PRZEJAZD
'------------------------
'W29.8
'------------------------
MOVL C00185 BC00185 V=500.0
SFTON P0302
MOVL C00186 BC00186 V=66.7 PL=0
MACRO1 MJ#(0) ARGF24
ARCON
MOVL C00187 BC00187 V=10.0
ARCOF
SFTOF
MOVL C00188 BC00188 V=500.0
SFTOF
MOVL C00189 BC00189 V=500.0
'PRZEJAZD
MOVL C00190 BC00190 V=500.0
MOVJ C00191 BC00191 VJ=20.00
MOVJ C00192 BC00192 VJ=10.00
MOVJ C00193 BC00193 VJ=10.00
'TEST
'TEST
'TEST
'TEST
'TEST
MOVJ C00194 BC00194 VJ=10.00
MOVJ C00195 BC00195 VJ=10.00
'------------------------
'W29.2
'------------------------
'PRZEJAZD
'------------------------
'W63.5
'------------------------
MOVL C00196 BC00196 V=500.0
SFTON P0351
MOVL C00197 BC00197 V=66.7 PL=0
MACRO1 MJ#(0) ARGF24
ARCON
MOVL C00198 BC00198 V=10.8
ARCOF
SFTOF
MOVL C00199 BC00199 V=500.0
'PRZEJAZD
MOVL C00200 BC00200 V=500.0
MOVL C00201 BC00201 V=500.0
MOVL C00202 BC00202 V=500.0
MOVL C00203 BC00203 V=500.0
'------------------------
'W29.8
'------------------------
MOVL C00204 BC00204 V=500.0
SFTON P0352
MOVL C00205 BC00205 V=66.7 PL=0
MACRO1 MJ#(0) ARGF24
ARCON
MOVL C00206 BC00206 V=10.8
ARCOF
SFTOF
MOVL C00207 BC00207 V=500.0
SFTOF
MOVL C00208 BC00208 V=500.0
'PRZEJAZD
MOVL C00209 BC00209 V=500.0
MOVJ C00210 BC00210 VJ=10.00
MOVJ C00211 BC00211 VJ=10.00
MOVJ C00212 BC00212 VJ=30.00
MOVJ C00213 BC00213 VJ=30.00
MOVJ C00214 BC00214 VJ=10.00
MOVJ C00215 BC00215 VJ=10.00
'------------------------
'W29.11
'------------------------
MOVL C00216 BC00216 V=500.0
MOVL C00217 BC00217 V=66.7
SFTON P0303
MOVL C00218 BC00218 V=66.7 PL=0
MACRO1 MJ#(0) ARGF24
ARCON
MOVL C00219 BC00219 V=10.8
ARCOF
SFTOF
MOVL C00220 BC00220 V=66.7
'PRZEJAZD
MOVL C00221 BC00221 V=500.0
MOVJ C00222 BC00222 VJ=10.00
MOVL C00223 BC00223 V=500.0
MOVL C00224 BC00224 V=500.0
'------------------------
'W29.14
'------------------------
MOVL C00225 BC00225 V=66.7
SFTON P0304
MOVL C00226 BC00226 V=66.7 PL=0
MACRO1 MJ#(0) ARGF24
ARCON
MOVL C00227 BC00227 V=10.8
ARCOF
SFTOF
MOVL C00228 BC00228 V=66.7
SFTOF
'PRZEJAZD
MOVL C00229 BC00229 V=500.0
MOVL C00230 BC00230 V=500.0
'------------------------
'W63.17
'------------------------
MOVL C00231 BC00231 V=66.7
SFTON P0305
MOVL C00232 BC00232 V=66.7 PL=0
MACRO1 MJ#(0) ARGF24
ARCON
MOVL C00233 BC00233 V=10.8
ARCOF
SFTOF
MOVL C00234 BC00234 V=66.7
MOVL C00235 BC00235 V=666.7
SFTOF
'PRZEJAZD
MOVJ C00236 BC00236 VJ=10.00
MOVJ C00237 BC00237 VJ=10.00
MOVJ C00238 BC00238 VJ=10.00
'COMMENT
'COMMENT
'COMMENT
'COMMENT
'COMMENT
MOVJ C00239 BC00239 VJ=10.00
MOVJ C00240 BC00240 VJ=10.00
MOVJ C00241 BC00241 VJ=10.00
MOVJ C00242 BC00242 VJ=10.00
'------------------------
'W28.11
'------------------------
MOVL C00243 BC00243 V=500.0
MOVL C00244 BC00244 V=66.7
SFTON P0353
MOVL C00245 BC00245 V=66.7 PL=0
MACRO1 MJ#(0) ARGF24
ARCON
MOVL C00246 BC00246 V=10.8
ARCOF
SFTOF
MOVL C00247 BC00247 V=66.7
'PRZEJAZD
MOVL C00248 BC00248 V=500.0
MOVJ C00249 BC00249 VJ=10.00
MOVL C00250 BC00250 V=500.0
MOVL C00251 BC00251 V=500.0
'------------------------
'W28.14
'------------------------
MOVL C00252 BC00252 V=66.7
SFTON P0354
MOVL C00253 BC00253 V=66.7 PL=0
MACRO1 MJ#(0) ARGF24
ARCON
MOVL C00254 BC00254 V=10.8
ARCOF
SFTOF
MOVL C00255 BC00255 V=66.7
SFTOF
'PRZEJAZD
MOVL C00256 BC00256 V=500.0
MOVL C00257 BC00257 V=500.0
'------------------------
'W62.17
'------------------------
MOVL C00258 BC00258 V=66.7
SFTON P0355
MOVL C00259 BC00259 V=66.7 PL=0
MACRO1 MJ#(0) ARGF24
ARCON
MOVL C00260 BC00260 V=10.8
ARCOF
SFTOF
MOVL C00261 BC00261 V=66.7
SFTOF
'PRZEJAZD
MOVJ C00262 BC00262 VJ=10.00
MOVJ C00263 BC00263 VJ=10.00
MOVJ C00264 BC00264 VJ=20.00
MOVJ C00265 BC00265 VJ=10.00
MOVJ C00266 BC00266 VJ=20.00
MOVJ C00267 BC00267 VJ=20.00
MOVL C00268 BC00268 V=500.0
MOVL C00269 BC00269 V=500.0
'------------------------
'W63.20
'------------------------
MOVL C00270 BC00270 V=500.0
SFTON P0306
MOVL C00271 BC00271 V=66.7 PL=0
MACRO1 MJ#(0) ARGF24
ARCON
MOVL C00272 BC00272 V=10.8
ARCOF
SFTOF
MOVL C00273 BC00273 V=500.0
'PRZEJAZD
MOVL C00274 BC00274 V=500.0
MOVL C00275 BC00275 V=500.0
MOVL C00276 BC00276 V=500.0
'------------------------
'W63.23
'------------------------
MOVL C00277 BC00277 V=500.0
SFTON P0307
MOVL C00278 BC00278 V=66.7 PL=0
MACRO1 MJ#(0) ARGF24
ARCON
MOVL C00279 BC00279 V=10.8
ARCOF
SFTOF
MOVL C00280 BC00280 V=500.0
SFTOF
'PRZEJAZD
'BRAK 29.26
'BRAK 29.26
'BRAK 29.26
'BRAK 29.26
'BRAK 29.26
'BRAK 29.26
MOVL C00281 BC00281 V=500.0
MOVJ C00282 BC00282 VJ=10.00
MOVJ C00283 BC00283 VJ=10.00
MOVJ C00284 BC00284 VJ=10.00
'TEST
'TEST
'TEST
'TEST
MOVJ C00285 BC00285 VJ=10.00
MOVJ C00286 BC00286 VJ=10.00
MOVJ C00287 BC00287 VJ=10.00
MOVL C00288 BC00288 V=500.0
MOVL C00289 BC00289 V=500.0
'------------------------
'W63.20
'------------------------
MOVL C00290 BC00290 V=500.0
SFTON P0356
MOVL C00291 BC00291 V=66.7 PL=0
MACRO1 MJ#(0) ARGF24
ARCON
MOVL C00292 BC00292 V=10.8
ARCOF
SFTOF
MOVL C00293 BC00293 V=500.0
'PRZEJAZD
MOVL C00294 BC00294 V=500.0
MOVL C00295 BC00295 V=500.0
MOVL C00296 BC00296 V=500.0
'------------------------
'W63.23
'------------------------
MOVL C00297 BC00297 V=500.0
SFTON P0357
MOVL C00298 BC00298 V=66.7 PL=0
MACRO1 MJ#(0) ARGF24
ARCON
MOVL C00299 BC00299 V=10.8
ARCOF
SFTOF
MOVL C00300 BC00300 V=500.0
SFTOF
'PRZEJAZD
'BRAK 29.26
'BRAK 29.26
'BRAK 29.26
'BRAK 29.26
'BRAK 29.26
'BRAK 29.26
MOVL C00301 BC00301 V=500.0
MOVJ C00302 BC00302 VJ=10.00
MOVJ C00303 BC00303 VJ=20.00
MOVJ C00304 BC00304 VJ=20.00
MOVJ C00305 BC00305 VJ=30.00
MOVJ C00306 BC00306 VJ=20.00
MOVJ C00307 BC00307 VJ=10.00
'------------------------
'W29.29
'------------------------
MOVL C00308 BC00308 V=66.7
SFTON P0309
MOVL C00309 BC00309 V=66.7 PL=0
MACRO1 MJ#(0) ARGF24
ARCON
MOVL C00310 BC00310 V=10.8
ARCOF
SFTOF
MOVL C00311 BC00311 V=66.7
SFTOF
'PRZEJAZD
MOVL C00312 BC00312 V=500.0
MOVJ C00313 BC00313 VJ=10.00
MOVJ C00314 BC00314 VJ=10.00
MOVJ C00315 BC00315 VJ=30.00
MOVJ C00316 BC00316 VJ=30.00
MOVJ C00317 BC00317 VJ=30.00
MOVJ C00318 BC00318 VJ=20.00
MOVL C00319 BC00319 V=333.3
'------------------------
'W29.29
'------------------------
MOVL C00320 BC00320 V=166.7
SFTON P0359
MOVL C00321 BC00321 V=166.7 PL=0
MACRO1 MJ#(0) ARGF24
ARCON
MOVL C00322 BC00322 V=10.8
ARCOF
SFTOF
MOVL C00323 BC00323 V=250.0
SFTOF
'PRZEJAZD
MOVL C00324 BC00324 V=500.0
'------------------------
'W29.32
'------------------------
MOVJ C00325 BC00325 VJ=30.00
MOVJ C00326 BC00326 VJ=40.00
MOVJ C00327 BC00327 VJ=40.00
MOVJ C00328 BC00328 VJ=30.00
CALL JOB:MOVE_OUT_OF_TUNNEL
END
